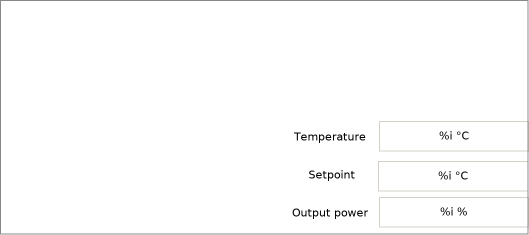
VISUALIZATION SerialCommVisuTest_1  // 529x235
    Textfield (379,121 150x30), "%i °C", text variable: SerialCommunicationController.pumpingPressureMeasurement
    Label (259,115 142x44), "Temperature"
    Label (259,191 142x44), "Output power"
    Textfield (379,197 150x30), "%i %", text variable: SerialCommunicationController.pumpingPressureOutputPower
    Textfield (378,161 150x30), "%i °C", text variable: SerialCommunicationController.pumpingPressureSetpoint
        OnMouseDown: write SerialCommunicationController.pumpingPressureSetSetpoint via VisuDialogs.Numpad, min 0, max 120
    Label (261,153 142x44), "Setpoint"
END_VISUALIZATION

(* stored: Version 1.1.0.1, ProductVersion 3.1.4024.9
   Visu SerialCommVisuTest_1: Id {9e230aac-ab98-4b32-b82c-f1c1a65b220f} *)
